Staubli VAL3: remGetRobotMode.pgx

program remGetRobotMode(string& sReturn[] (dimensions=1))
  local string sCmd
begin
  // Return the PPS status saved in the robot
  //
  logMsg("call remGetRobotMode")
  sCmd="GETROBOTMODE"
  call remGetnGlobal(nRobotMode,sCmd,sReturn)
end
